PROGRAM MAIN
VAR
	AxisBaseObject : BaseModuleToBeVisited(MyName := 'axis1');
	Status : T_MaxString := '';
	statusStringVisitor : StatusToStringLogVisitor(Status);
	RunStatusReport: BOOL;
END_VAR

END_PROGRAM

(* stored: Version 1.1.0.1, ProductVersion 3.1.4024.12
   POU MAIN: Id {94e20353-7e7b-4773-9ab6-97fa33344c4a}, SpecialFunc None *)
